FUNCTION TryConvert_TOD_TO_LWORD : BOOL
VAR_INPUT
	in : TOD;
	out : REFERENCE TO LWORD;
END_VAR

out := TOD_TO_LWORD(in);
TryConvert_TOD_TO_LWORD := TRUE;

END_FUNCTION

(* stored: Version 1.1.0.1, ProductVersion 3.1.4024.12
   POU TryConvert_TOD_TO_LWORD: Id {734ea458-0dca-420f-9585-d04fbcb06600}, SpecialFunc None *)
